{attribute 'qualified_only'}
VAR_GLOBAL
//INT
	NO					:	INT		;
//Bool
	Status				:	BOOL	;
	Vision_Start		:	BOOL	;
	Wait_Vision_OK		:	BOOL	;
	Data_Copy: BOOL;
	Data_Initial: BOOL;
	Data_Copy_Check: BOOL;
END_VAR

(* stored: Version 1.1.0.1, ProductVersion 3.1.4024.15
   GVL GVL_Vision_Step: Id {a62b2c31-2e11-4b06-b4e9-cefa61950d78} *)
